TYPE ST_APP_CTRL :
STRUCT
  Cmd       : E_INSTANCE_CMD;
END_STRUCT
END_TYPE

(* stored: Version 1.1.0.1, ProductVersion 3.1.4024.15
   DUT ST_APP_CTRL: Id {df31154c-b784-4bef-8cca-12faddca3455} *)
